FUNCTION_BLOCK FB_FastDoorAddon EXTENDS FB_FunctionConv
VAR_INPUT
	Config						: ST_CFG_FastDoor; 		// Configuration
	HW_Inputs					: ST_HW_InputsFastDoor; 	// Hardware inputs
END_VAR

VAR_OUTPUT	
	HW_Outputs					: ST_HW_OutputsFastDoor; // Hardware outputs
END_VAR

VAR
	Inputs						: ST_InputsFastDoor;  // Function specific inputs
	Outputs						: ST_OutputsFastDoor; // Function specific outputs  
	fbAddonErrHandler			: FB_AddOnErrHandler;
	FastDoorStates				: ST_FastDoorStates;
	FastDoorData				: ST_FastDoorData; 
END_VAR

VAR PERSISTENT
	Settings					: ST_CFG_FastDoor; // Settings - activated configuration 
END_VAR

(**************************************************************************************************************
   Input mapping
***************************************************************************************************************)
A_InputMapping();

(**************************************************************************************************************
   Initialization
***************************************************************************************************************)
A_Init();

(**************************************************************************************************************
  BCF State control
***************************************************************************************************************)
A_StateControl();

(**************************************************************************************************************
   Error handler
***************************************************************************************************************)
A_ErrorHandler();
fbAddOnErrHandler(AddOnSettingsFunction :=SettingsFunction, AddOnFunctionData:=FunctionData);
_M_CheckErrors();

(**************************************************************************************************************
   Process AddOns
***************************************************************************************************************)
M_ProcessAddOns();

(**********************************************************************************************************
   State Handler 
***********************************************************************************************************)
_M_FastDoorStates();

(**********************************************************************************************************
   Control Door 
***********************************************************************************************************)
_M_ControlDoor(); 

(**********************************************************************************************************
   Check Error 
***********************************************************************************************************)
_M_CheckErrors();

(**************************************************************************************************************
   Interface handler out
***************************************************************************************************************)
M_ITC_ProcessOut();

(**************************************************************************************************************
   Output mapping
***************************************************************************************************************)
A_OutputMapping();

METHOD PRIVATE _M_CheckErrors : BOOL
VAR_INPUT 
END_VAR

VAR
END_VAR
F_ResetError(FALSE,	FunctionData.ErrorData.ErrorDataSet[2]);

IF NOT Inputs.HW.Ready THEN 
	F_SetError(
		ErrorType 	:= E_ErrorType.ERROR,
		ErrorParam 	:= 'Door ready signal not set',
		ErrorMsg 	:= E_ErrorConv.DOOR_ERROR,
		ErrorData 	:= FunctionData.ErrorData.ErrorDataSet[2]);	
END_IF
END_METHOD

METHOD PRIVATE _M_ControlDoor : BOOL

VAR
	fbDoorOpenTrigger	: R_TRIG;
END_VAR

_M_DoorControl(
	SensorPosDown:= Inputs.HW.Closed, 
	SensosPosUp:= Inputs.HW.Open, 
	TimeOutValueDoor:= Settings.TimeoutValueDoor, 
	OrderPos:= FastDoorData.OrderPos,  
	DriveUp=> Outputs.HW.OpenDoor, 
	DriveDown=> Outputs.HW.CloseDoor, 
	EnableTransport=> FastDoorData.EnableTransport);
END_METHOD

METHOD PRIVATE _M_DoorControl : BOOL
VAR_INPUT
	SensorPosDown		: BOOL;
	SensosPosUp			: BOOL; 
	TimeOutValueDoor	: TIME;
	OrderPos			: E_DoorPos;
END_VAR

VAR_OUTPUT
	DriveUp				: BOOL; 
	DriveDown			: BOOL;
	EnableTransport		: BOOL; 
END_VAR

VAR_INST
	eState				: E_FastDoorControlStates;
	eLastState			: E_FastDoorControlStates;
	fbTimeoutTimer		: TON;
END_VAR
F_ResetError(FALSE,	FunctionData.ErrorData.ErrorDataSet[1]);

fbTimeoutTimer.IN := FALSE;
fbTimeoutTimer.PT := TimeOutValueDoor;

CASE eState	OF 
	
	(**************************************************************************************************************
 	INIT
	***************************************************************************************************************)
	E_FastDoorControlStates.INIT:
		DriveUp := FALSE;
		DriveDown := FALSE;
		EnableTransport := FALSE;
		
		eLastState := eState;
		eState := E_FastDoorControlStates.IDLE;	

	(**************************************************************************************************************
 	IDLE
	***************************************************************************************************************)
	E_FastDoorControlStates.IDLE:
		
		IF OrderPos = E_DoorPos.DOWN THEN
		
			IF SensorPosDown THEN
				EnableTransport := TRUE;
			ELSE
				EnableTransport := FALSE;
				eLastState := eState;
				eState := E_FastDoorControlStates.DOOR_DOWN;
			END_IF
		
		ELSIF OrderPos  = E_DoorPos.UP THEN
			IF SensosPosUp THEN
				EnableTransport := TRUE;
			ELSE
				EnableTransport := FALSE;
				eLastState := eState;
				eState := E_FastDoorControlStates.DOOR_UP;
			END_IF
		ELSE
			EnableTransport := FALSE; 
		END_IF
					
	(**************************************************************************************************************
 	DOOR_DOWN
	***************************************************************************************************************)
	E_FastDoorControlStates.DOOR_DOWN:
	
		IF SensorPosDown THEN 
			DriveDown := FALSE;
			eLastState := eState; 
			eState := E_FastDoorControlStates.IDLE;
		ELSE
			fbTimeoutTimer.IN := TRUE;
			
			IF fbTimeoutTimer.Q THEN 
				F_SetError(
					ErrorType	:= E_ErrorType.ERROR,
					ErrorParam	:= 'Timeout closing door',
					ErrorMsg 	:= E_ErrorConv.TIMEOUT_MOVEMENT,
					ErrorData	:= FunctionData.ErrorData.ErrorDataSet[1]);
			ELSE
				DriveDown := TRUE;
			END_IF
		END_IF

	(**************************************************************************************************************
 	DOOR_UP
	***************************************************************************************************************)
	E_FastDoorControlStates.DOOR_UP:
	
		IF SensosPosUp THEN 
			DriveUp := FALSE;
			eLastState := eState; 
			eState := E_FastDoorControlStates.IDLE;
			
		ELSE
			fbTimeoutTimer.IN := TRUE; 
			
			IF fbTimeoutTimer.Q THEN
				F_SetError(
					ErrorType	:= E_ErrorType.ERROR,
					ErrorParam	:= 'Timeout opening door',
					ErrorMsg 	:= E_ErrorConv.TIMEOUT_MOVEMENT,
					ErrorData	:= FunctionData.ErrorData.ErrorDataSet[1]);
			ELSE
				DriveUp := TRUE; 
			END_IF
			
		END_IF
END_CASE

//Call timer 
fbTimeoutTimer();
END_METHOD

METHOD PRIVATE _M_DoorSide : BOOL
VAR_INPUT
	TrspData					: REFERENCE TO ST_TransportControlData;
	TrspDataNext				: REFERENCE TO ST_TransportControlData;
	TrspDataPrev				: REFERENCE TO ST_TransportControlData;
	Side						: INT; 
END_VAR

VAR
	AdjacentSide				: E_FunctionNumber;
END_VAR

VAR_IN_OUT
	Error		: ST_ErrorDataSet;  
END_VAR
IF NOT __ISVALIDREF(FunctionRegistry[SettingsFunction.FunctionLink.eFunctionNumber].rFunctionInterface) THEN 
	RETURN;
END_IF

IF NOT __ISVALIDREF(FunctionRegistry[SettingsFunction.FunctionLink.eFunctionNumber].rSettingsFunction) THEN 
	RETURN;
END_IF

IF NOT (Side > 0 AND Side <= 4) THEN
	F_SetError(
			ErrorType	:= E_ErrorType.ERROR,
			ErrorParam	:= 'Door side number not defined',
			ErrorMsg 	:= E_ErrorConv.CONFIGURATION_ERROR,
			ErrorData	:= Error);
END_IF

AdjacentSide := FunctionRegistry[SettingsFunction.FunctionLink.eFunctionNumber].rSettingsFunction.eAdjacentFunctionNumberSide[Side];

IF(( FunctionRegistry[SettingsFunction.FunctionLink.eFunctionNumber].rFunctionInterface.In.eNextFunctionNumber = AdjacentSide AND 
	TrspData.NumberOfPresentTUs > 0) OR
	(FunctionRegistry[SettingsFunction.FunctionLink.eFunctionNumber].rFunctionInterface.In.ePrevFunctionNumber = AdjacentSide AND
	TrspData.NumberOfPresentTUs = 0)) THEN
	
	_M_DoorSide := TRUE;
END_IF
END_METHOD

METHOD _M_FastDoorStates : BOOL

VAR
	TrspData					: ST_TransportControlData;
	TrspDataNext				: ST_TransportControlData;
	TrspDataPrev				: ST_TransportControlData;
	ZoneIndexNext				: INT;
	ZoneIndexPrev				: INT; 
END_VAR

VAR_INST
	fbTimerWait		: TON;
END_VAR
F_ResetError(FALSE,	FunctionData.ErrorData.ErrorDataSet[1]);

TrspData := F_PB_GetTransportControlDataRef(eFunctionNumber	:= SettingsFunction.FunctionLink.eFunctionNumber,
											ZoneNumber := SettingsFunction.FunctionLink.ZoneNumber);
											
F_PB_GetAdjacentFunctionZoneIndex(	CheckFunction:= SettingsFunction.FunctionLink.eFunctionNumber, 
									ExpectedFunction:= FunctionRegistry[SettingsFunction.FunctionLink.eFunctionNumber].rFunctionInterface.In.eNextFunctionNumber, 
									RequireNextDefined:= TRUE, 
									RequirePreviousDefined:= FALSE, 
									ZoneIndex:= ZoneIndexNext);								
													
TrspDataNext := F_PB_GetTransportControlDataRef(eFunctionNumber	:= FunctionRegistry[SettingsFunction.FunctionLink.eFunctionNumber].rFunctionInterface.In.eNextFunctionNumber,
												ZoneNumber 	:= ZoneIndexNext);
												
F_PB_GetAdjacentFunctionZoneIndex(	CheckFunction:= SettingsFunction.FunctionLink.eFunctionNumber, 
									ExpectedFunction:= FunctionRegistry[SettingsFunction.FunctionLink.eFunctionNumber].rFunctionInterface.In.ePrevFunctionNumber, 
									RequireNextDefined:= FALSE, 
									RequirePreviousDefined:= TRUE, 
									ZoneIndex:= ZoneIndexPrev);								
													
TrspDataPrev := F_PB_GetTransportControlDataRef(eFunctionNumber	:= FunctionRegistry[SettingsFunction.FunctionLink.eFunctionNumber].rFunctionInterface.In.ePrevFunctionNumber,
												ZoneNumber 	:= ZoneIndexPrev);

FastDoorData.DoorSide := _M_DoorSide(TrspData, TrspDataNext, TrspDataPrev, Settings.DoorSide, FunctionData.ErrorData.ErrorDataSet[1]);

fbTimerWait.IN := FALSE; 
fbTimerWait.PT := Settings.WaitTime;

CASE FastDoorStates.eState OF
(**************************************************************************************************************
 INIT
***************************************************************************************************************)
	E_FastDoorState.INIT:
	
	fbTimerWait.IN := FALSE;
	Outputs.HW.KeepDoorOpen := FALSE;
	
	FastDoorStates.eLastState := FastDoorStates.eState;
	FastDoorStates.eState := E_FastDoorState.CLOSED;

		
(**************************************************************************************************************
 CLOSED
***************************************************************************************************************)
	E_FastDoorState.CLOSED:
	
	fbTimerWait.IN := FALSE;
	Outputs.HW.KeepDoorOpen := FALSE;
	
	FastDoorData.OrderPos := E_DoorPos.DOWN;

	//Check if transport is on side with door or not
	//False also when Next or Prev function is not set
	IF FastDoorData.DoorSide THEN
		
		IF( TrspData.NumberOfPresentTUs > 0 AND TrspDataNext.NumberOfPresentTUs = 0) OR
		  ( TrspData.NumberOfPresentTUs = 0 AND TrspDataPrev.NumberOfPresentTUs > 0) THEN
		  
			//Change state
			FastDoorStates.eLastState := FastDoorStates.eState;
			FastDoorStates.eState := E_FastDoorState.OPENING;
		END_IF
	END_IF
	
(**************************************************************************************************************
 OPENING
***************************************************************************************************************)
	E_FastDoorState.OPENING:
	
	FastDoorData.OrderPos := E_DoorPos.UP;
	
	//When door is opened
	IF Inputs.HW.Open THEN
		
		//Change state
		FastDoorStates.eLastState := FastDoorStates.eState;
		FastDoorStates.eState := E_FastDoorState.OPEN;
	END_IF
	
(**************************************************************************************************************
 OPEN
***************************************************************************************************************)
	E_FastDoorState.OPEN:
	
	fbTimerWait.IN := TRUE;

	IF fbTimerWait.Q THEN
		//Change state
		FastDoorStates.eLastState := FastDoorStates.eState;
		FastDoorStates.eState := E_FastDoorState.CLOSED;
	END_IF
	
	IF FastDoorData.DoorSide THEN
		
		IF( TrspData.NumberOfPresentTUs > 0 AND TrspDataNext.NumberOfPresentTUs = 0) OR
		  ( TrspData.NumberOfPresentTUs = 0 AND TrspDataPrev.NumberOfPresentTUs > 0) THEN
		  
			Outputs.HW.KeepDoorOpen := TRUE;
			fbTimerWait.IN := FALSE;
			
		END_IF 
	END_IF
END_CASE

//Call timer 
fbTimerWait();
END_METHOD

ACTION A_Init:
(**************************************************************************************
 * 	NAME		A_Init
 * 	FUNCTION	Initialize function
 **************************************************************************************)
 
// Update Registry
M_UpdateRegistry();


// Init ongoing - Wait until init is released (Sequencial startup)
IF NOT FunctionData.Init AND FunctionData.InitRunning THEN
	// When the subsystem is started, 
	// When its released to initialize
	IF FunctionData.OperationState.Info.SystemReady AND
	   SettingsFunction.eFunctionNumber < FunctionData.OperationState.InitRelease.eLimitFunctionNumber THEN
	   
	   IF M_InitFunction(FALSE) THEN		   
			// Function initialized - and initialization done
			FunctionData.Init := TRUE;
			FunctionData.InitRunning := FALSE;
			
			FastDoorStates.eLastState := FastDoorStates.eState;
			FastDoorStates.eState := E_FastDoorState.INIT;
			
			// Set reset cmd
			FunctionData.ErrorData.Error.ResetError := TRUE;
			
			DebugMsg := CONCAT('Initialization done. Function: ', ConfigFunction.FunctionName);
			fbDebugMsg.M_SendInfoMsg(DebugMsg);
		END_IF
	END_IF
(*
If the function is not initialized,
clean all values and wait until init is released
*)
ELSIF NOT FunctionData.Init THEN
	// Reset internal variables
	FunctionData.OperationState := FunctionBase.PositionStateEmpty;

	// Initiate initialization of all zones
	(*FOR ZoneIdx := 1 TO SettingsFunction.NumberOfZones DO
		ZoneData[ZoneIdx].Init := FALSE;
	END_FOR;*)
	
	// Load function specific configuration to settings
	Settings := Config;
	
	// Reset values and load config
	M_PreInit();	
	
	// To start init a valid functionnumber and element link is needed
	FunctionData.InitRunning := SettingsFunction.eFunctionNumber > 0 AND
								SettingsFunction.eElementLink > 0;
								
								
END_IF
END_ACTION

ACTION A_InputMapping:
(**************************************************************************************
 * 	NAME		A_InputMapping
 * 	FUNCTION	Input mapping
 **************************************************************************************)
 
(**************************************************************************************
   Hardware Inputs
***************************************************************************************)

Inputs.HW := HW_Inputs;

(**************************************************************************************
   Element states
***************************************************************************************)
// Get status of the corresponding element
M_GetElementStates();
END_ACTION

ACTION A_OutputMapping:
(**************************************************************************************
 * 	NAME		A_OutputMapping
 * 	FUNCTION	Output mapping
 **************************************************************************************)
 
(**************************************************************************************
   Hardware outputs
***************************************************************************************)
HW_Outputs.CloseDoor			:= Outputs.HW.CloseDoor;
HW_Outputs.KeepDoorOpen			:= Outputs.HW.KeepDoorOpen;
HW_Outputs.OpenDoor				:= Outputs.HW.OpenDoor;
HW_Outputs.StopDrive			:= Outputs.HW.StopDrive; 
		
(**************************************************************************************
   Order outputs (Commands to corresponding element)
***************************************************************************************)
MEMSET(ADR(FunctionInterface.Out.FunctionOrders),0,SIZEOF(ST_FunctionOrders));
FunctionInterface.Out.FunctionOrders.Enable 				:= FunctionData.ErrorData.Error.ErrorType = E_ErrorType.NO_ERROR_PENDING;

(**************************************************************************************
   AddOn outputs
***************************************************************************************)

FunctionInterface.Out.AddOnOrders.Enable 					:= FunctionData.ErrorData.Error.ErrorType <> E_ErrorType.ERROR;
FunctionInterface.Out.AddOnOrders.DataReady					:= TRUE;

IF FastDoorData.DoorSide THEN
	FunctionInterface.Out.AddOnOrders.EnableHandover 			:= FastDoorData.EnableTransport AND Inputs.HW.Open;
	FunctionInterface.Out.AddOnOrders.EnableTakeover 			:= FastDoorData.EnableTransport AND Inputs.HW.Open;
ELSE
	FunctionInterface.Out.AddOnOrders.EnableHandover 			:= TRUE;
	FunctionInterface.Out.AddOnOrders.EnableTakeover 			:= TRUE;
END_IF


(**************************************************************************************
   Status outputs
***************************************************************************************)

//Inhibit stopping for the function when ExtendedRun is driving
THIS^.InhibitStopping := NOT FastDoorData.EnableTransport;
END_ACTION

END_FUNCTION_BLOCK

(* stored: Version 1.1.0.1, ProductVersion 3.1.4024.9
   POU FB_FastDoorAddon: Id {77b33f93-001a-4c35-8a63-7df432e36bc8}, SpecialFunc None
   Method _M_CheckErrors: Id {8b99d517-5ceb-4686-a8d8-4ea4e690d79d}
   Method _M_ControlDoor: Id {62810f2d-077b-4b83-8f06-e2fd4f93ef5e}
   Method _M_DoorControl: Id {89384305-67e4-4f50-9684-c42688dff6b0}
   Method _M_DoorSide: Id {8b71b0b1-4444-43c3-ae8f-bf4c82dbd50e}
   Method _M_FastDoorStates: Id {5e91031c-efa6-481f-a3b5-00babbaa528e}
   Action A_Init: Id {2c56a7fa-2048-4bcd-a7e2-816174a123e2}
   Action A_InputMapping: Id {7b66e336-85a3-4313-8d5c-348bf5a65066}
   Action A_OutputMapping: Id {58d4c10a-1932-49a1-9989-a7a136362c5b} *)
